(* PLC project test_order, GEENSOFT ControlBuild 2010-3c *)
(* stored: creationDateTime 2011-09-14T10:40:23-01:00 *)

FUNCTION_BLOCK hvs.test_order
  VAR_INPUT
    Test2 : BOOL := false;
  END_VAR
  VAR_INPUT
    Test1 : BOOL := false;
  END_VAR
  VAR_INPUT
    A1 : BOOL := false;
    A2 : BOOL := false;
    A3 : BOOL := false;
    A4 : BOOL := false;
  END_VAR
  VAR_INPUT
    A22 : BOOL := false;
    B : BOOL := false;
    D : BOOL := false;
    E : BOOL := false;
  END_VAR
  VAR_OUTPUT
    Test5 : BOOL := false;
  END_VAR
  VAR_OUTPUT
    Test3 : BOOL := false;
  END_VAR
  VAR_OUTPUT
    A5 : BOOL := false;
    A6 : BOOL := false;
    A7 : BOOL := false;
    A9 : BOOL := false;
  END_VAR
  VAR_OUTPUT
    A11 : BOOL := false;
    A12 : BOOL := false;
    A13 : BOOL := false;
    A14 : BOOL := false;
    B1 : BOOL := false;
    D1 : BOOL := false;
    E1 : BOOL := false;
    Test4 : BOOL := false;
    Test6 : BOOL := false;
  END_VAR

(* FBD diagram, written out as Structured Text *)
END_FUNCTION_BLOCK
